(* Logix 5000 project; controller GEA_Test_Chamber vendor 1 type 14 code 196 rev 32.14; software revision 32.04; part 10 of 11 *)
(* tags used below, declared in another part *)
   bPulse1Hz : BOOL;
   Counter : COUNTER[20];
   LDO_LabView_Comm_OK : BOOL;
   LDO_Step : INT;
   LDO_Timer_Delay : TIMER[30];
   LDO_Water_Outlet_HighLimit : REAL;
   LDO_Water_Outlet_LowLimit : REAL;
   Oil_spray_11_ccmin : BOOL;
   ONS : BOOL[32];
   test : BOOL;
   Water_Outlet_Temp_OK : BOOL;
   Amount_Water_Flow : DINT;
   Client_01 : raC_Opr_NetModbusTCPClient;
   Client_01_Data : raC_UDT_ModbusClientData;
   Client_01_EN : BOOL;
   Client_01_MSG_Connect : MESSAGE;
   Client_01_MSG_Create : MESSAGE;
   Client_01_MSG_Delete : MESSAGE;
   Client_01_MSG_Read : MESSAGE;
   Client_01_MSG_SetSing : MESSAGE;
   Client_01_MSG_Write : MESSAGE;
   Client_01_Parameters : raC_UDT_ModbusClientConnection;
   Client_01_Transactions : raC_UDT_ModbusClientTransaction[5];
   Client_02 : raC_Opr_NetModbusTCPClient;
   Client_02_Data : raC_UDT_ModbusClientData;
   Client_02_EN : BOOL;
   Client_02_MSG_Connect : MESSAGE;
   Client_02_MSG_Create : MESSAGE;
   Client_02_MSG_Delete : MESSAGE;
   Client_02_MSG_Read : MESSAGE;
   Client_02_MSG_SetSing : MESSAGE;
   Client_02_MSG_Write : MESSAGE;
   Client_02_Parameters : raC_UDT_ModbusClientConnection;
   Client_02_Transactions : raC_UDT_ModbusClientTransaction[5];
   FVIR_Error_MSG : INT;
   FVIR_LabView_Control : INT;
   FVIR_LabView_Status : INT;
   FVIR_Mannequin_Direction_TimeDelay : INT;
   FVIR_Mannequin_Time_Pause : INT;
   FVIR_Number_Mannequin_Movement : INT;
   FVIR_Rate_REAL : REAL;
   FVIR_Reset_Cnt : BOOL;
   FVIR_Reset_Cnt_inprogress : BOOL;
   FVIR_Test_No : INT;
   FVIR_Totalizer_REAL : REAL;
   FVIR_Water_Flow_DRK375 : INT;
   FVIR_Water_Flow_DRK375_Float : REAL;
   FVIR_Water_Outlet_Valve : INT;
   FVIR_Water_Outlet_Valve_Flow_SP : REAL;
   FVIR_Water_Outlet_Valve_SP : REAL;
   FVIR_Water_Temp_DRK375 : INT;
   FVIR_Water_Temp_DRK375_Float : REAL;
   LDO_BurnerCycle_11_12_OFF : INT;
   LDO_BurnerCycle_11_12_ON : INT;
   LDO_BurnerCycle_13_OFF : INT;
   LDO_BurnerCycle_13_ON : INT;
   LDO_BurnerCycle_1_10_OFF : INT;
   LDO_BurnerCycle_1_10_ON : INT;
   LDO_Error_MSG : INT;
   LDO_LabView_Control : INT;
   LDO_LabView_Control2 : INT;
   LDO_LabView_Status : INT;
   LDO_Oil_1st_seq_OFF : INT;
   LDO_Oil_1st_seq_ON : INT;
   LDO_Oil_all_seq_OFF : INT;
   LDO_Oil_all_seq_ON : INT;
   LDO_Oil_pre_seq_OFF : INT;
   LDO_Oil_pre_seq_ON : INT;
   LDO_Reset_Cnt : BOOL;
   LDO_Reset_CNT_inprogress : BOOL;
   LDO_Water_Flow_DRK375_Float : REAL;
   LDO_Water_Outlet_Valve : REAL;
   LDO_Water_Outlet_Valve_Flow_SP : REAL;
   LDO_Water_Outlet_Valve_SP : REAL;
   LDO_Water_Temp_DRK375_Float : REAL;
   Modbus_LabView : raC_Opr_NetModbusTCPServer;
   Modbus_LabView_Data : raC_UDT_ModbusServerData;
   nLDO_Rate_REAL : REAL;
   nLDO_Totalizer_REAL : REAL;
   Output_LDO : Output_LDO;
   pulsReset : BOOL;
   SET_0 : BOOL;
   Timer_Delay_Start : TIMER;
(* LDO_Chamber, continued *)

ROUTINE LDO_Test   (* ladder *)
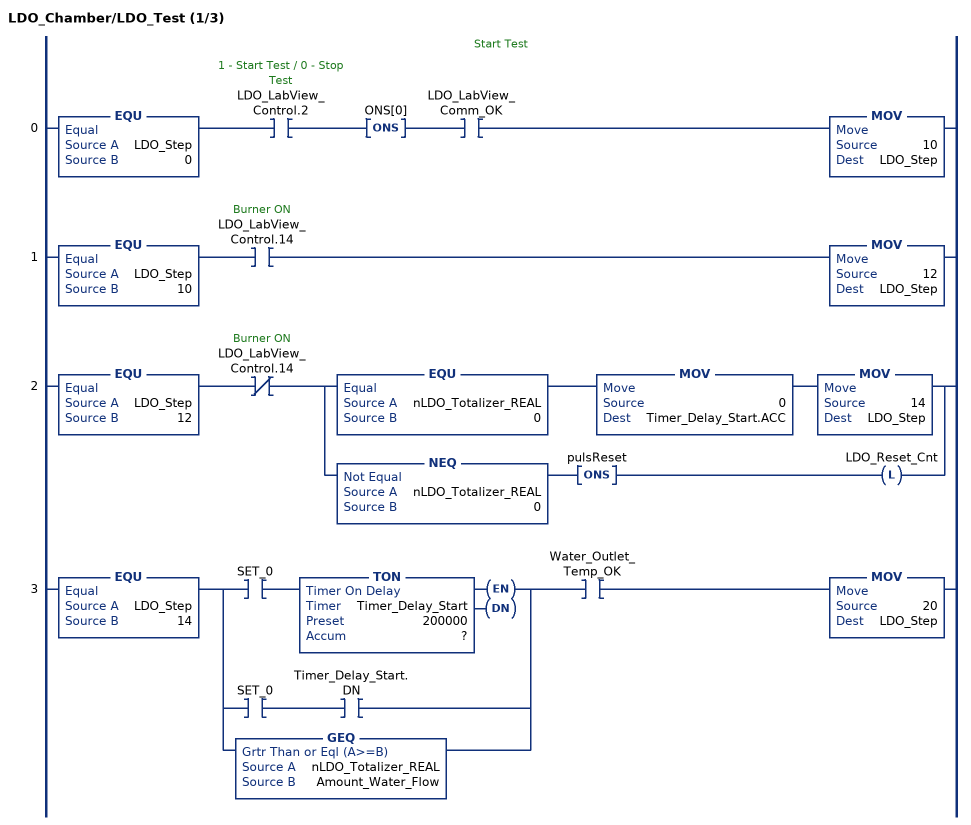
   // Start Test
   0: EQU(LDO_Step,0)XIC(LDO_LabView_Control.2)ONS(ONS[0])XIC(LDO_LabView_Comm_OK)MOV(10,LDO_Step);
   1: EQU(LDO_Step,10)XIC(LDO_LabView_Control.14)MOV(12,LDO_Step);
   2: EQU(LDO_Step,12)XIO(LDO_LabView_Control.14)[EQU(nLDO_Totalizer_REAL,0) MOV(0,Timer_Delay_Start.ACC) MOV(14,LDO_Step) ,NEQ(nLDO_Totalizer_REAL,0) ONS(pulsReset) OTL(LDO_Reset_Cnt) ];
   3: EQU(LDO_Step,14)[XIC(SET_0) TON(Timer_Delay_Start,?,?) ,XIC(SET_0) XIC(Timer_Delay_Start.DN) ,GEQ(nLDO_Totalizer_REAL,Amount_Water_Flow) ]XIC(Water_Outlet_Temp_OK)MOV(20,LDO_Step);
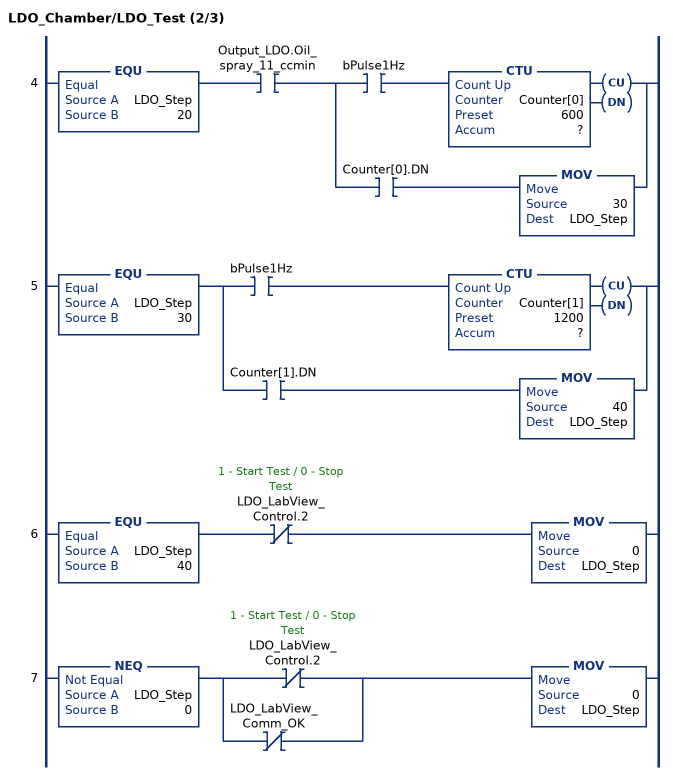
   4: EQU(LDO_Step,20)XIC(Output_LDO.Oil_spray_11_ccmin)[XIC(bPulse1Hz) CTU(Counter[0],?,?) ,XIC(Counter[0].DN) MOV(30,LDO_Step) ];
   5: EQU(LDO_Step,30)[XIC(bPulse1Hz) CTU(Counter[1],?,?) ,XIC(Counter[1].DN) MOV(40,LDO_Step) ];
   6: EQU(LDO_Step,40)XIO(LDO_LabView_Control.2)MOV(0,LDO_Step);
   7: NEQ(LDO_Step,0)[XIO(LDO_LabView_Control.2) ,XIO(LDO_LabView_Comm_OK) ]MOV(0,LDO_Step);
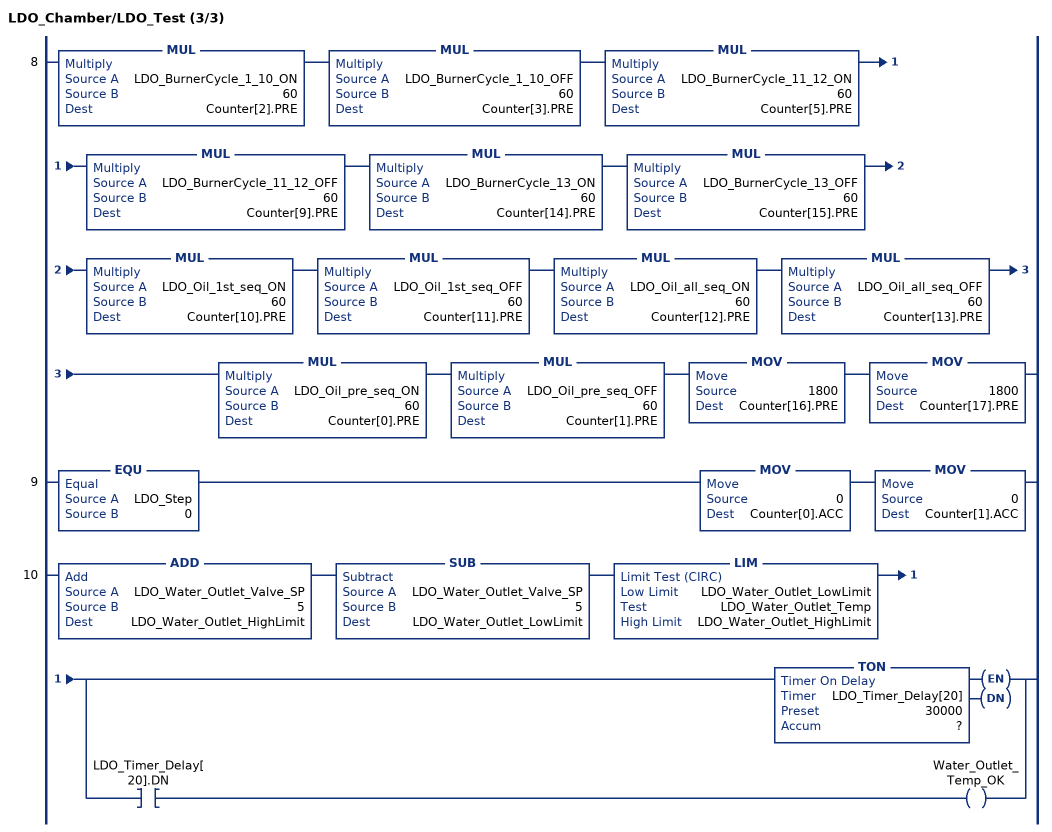
   8: MUL(LDO_BurnerCycle_1_10_ON,60,Counter[2].PRE)MUL(LDO_BurnerCycle_1_10_OFF,60,Counter[3].PRE)MUL(LDO_BurnerCycle_11_12_ON,60,Counter[5].PRE)MUL(LDO_BurnerCycle_11_12_OFF,60,Counter[9].PRE)MUL(LDO_BurnerCycle_13_ON,60,Counter[14].PRE)MUL(LDO_BurnerCycle_13_OFF,60,Counter[15].PRE)MUL(LDO_Oil_1st_seq_ON,60,Counter[10].PRE)MUL(LDO_Oil_1st_seq_OFF,60,Counter[11].PRE)MUL(LDO_Oil_all_seq_ON,60,Counter[12].PRE)MUL(LDO_Oil_all_seq_OFF,60,Counter[13].PRE)MUL(LDO_Oil_pre_seq_ON,60,Counter[0].PRE)MUL(LDO_Oil_pre_seq_OFF,60,Counter[1].PRE)MOV(1800,Counter[16].PRE)MOV(1800,Counter[17].PRE);
   9: EQU(LDO_Step,0)MOV(0,Counter[0].ACC)MOV(0,Counter[1].ACC);
   10: ADD(LDO_Water_Outlet_Valve_SP,5,LDO_Water_Outlet_HighLimit)SUB(LDO_Water_Outlet_Valve_SP,5,LDO_Water_Outlet_LowLimit)LIM(LDO_Water_Outlet_LowLimit,LDO_Water_Outlet_Temp,LDO_Water_Outlet_HighLimit)[TON(LDO_Timer_Delay[20],?,?) ,XIC(LDO_Timer_Delay[20].DN) OTE(Water_Outlet_Temp_OK) ];
END_ROUTINE
END_PROGRAM

PROGRAM Modbus_Client   (* main routine Main *)
VAR
   FVIR_Cnt_Reset : BOOL;
   FVIR_Rate_DINT : DINT;
   FVIR_Rate_value_temp : DINT;
   FVIR_Reset_Cnt_Timeout : TIMER := (PRE := 3000);
   FVIR_Reset_Cycle : DINT;
   FVIR_Timer_Delay_Reset : TIMER := (PRE := 500);
   FVIR_Timer_Reset : TIMER := (PRE := 500);
   FVIR_Total_DINT : DINT;
   FVIR_Total_value_temp : DINT;
   LDO_Cnt_Reset : BOOL;
   LDO_Rate_DINT : DINT;
   LDO_Rate_REAL : REAL;
   LDO_Rate_value_temp : DINT;
   LDO_Total_value_temp : DINT := 124780544;
   LDO_Totalizer_DINT : DINT := 1904;
   LDO_Totalizer_REAL : REAL := 4.91;
   LDO_Valley_value : DINT := 2034;
   LDO_Valley_value_temp : DINT := 133300224;
   Modbus_FVIR_Off : BOOL := 1;
   nLDO_Total_Mem : REAL := 565.7;
   off : BOOL := 1;
   ONS_1 : BOOL := 1;
   ONS_2 : BOOL;
   Reset_Cnt_Timeout : TIMER := (PRE := 3000);
   Reset_Cycle : DINT;
   Timer_Delay_Reset : TIMER := (PRE := 500);
   Timer_Reset : TIMER := (PRE := 500);
END_VAR

ROUTINE FVIR_Flow_Outlet_Meter   (* ladder *)
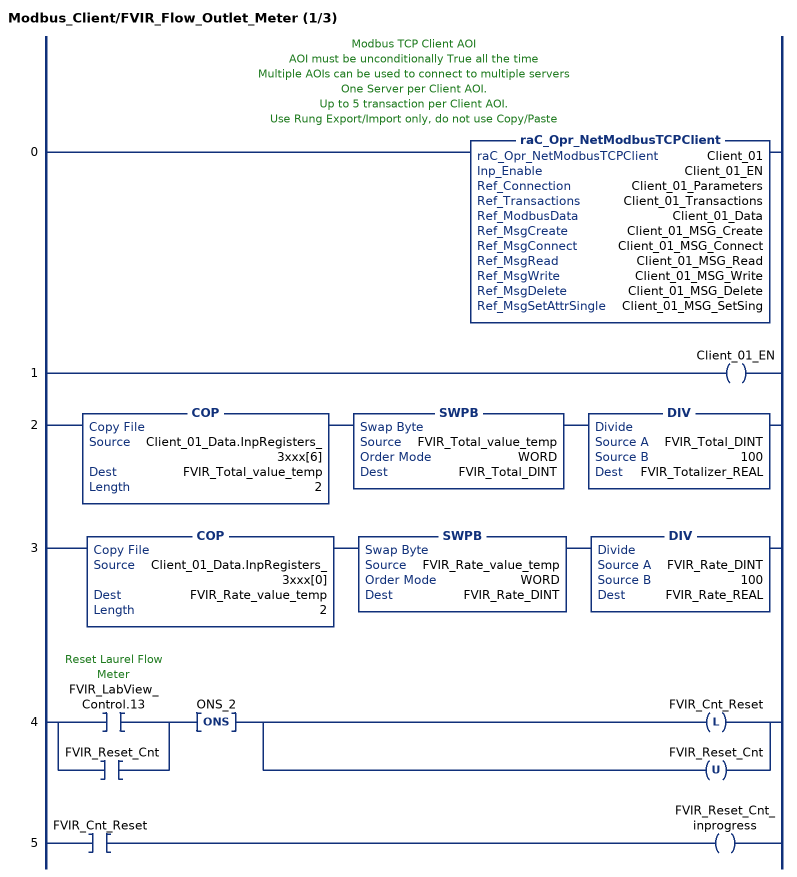
   // Modbus TCP Client AOI
   // AOI must be unconditionally True all the time
   // Multiple AOIs can be used to connect to multiple servers
   // One Server per Client AOI.
   //  Up to 5 transaction per Client AOI.
   // Use Rung Export/Import only, do not use Copy/Paste
   0: raC_Opr_NetModbusTCPClient(Client_01,Client_01_EN,Client_01_Parameters,Client_01_Transactions,Client_01_Data,Client_01_MSG_Create,Client_01_MSG_Connect,Client_01_MSG_Read,Client_01_MSG_Write,Client_01_MSG_Delete,Client_01_MSG_SetSing);
   1: OTE(Client_01_EN);
   2: COP(Client_01_Data.InpRegisters_3xxx[6],FVIR_Total_value_temp,2)SWPB(FVIR_Total_value_temp,WORD,FVIR_Total_DINT)DIV(FVIR_Total_DINT,100,FVIR_Totalizer_REAL);
   3: COP(Client_01_Data.InpRegisters_3xxx[0],FVIR_Rate_value_temp,2)SWPB(FVIR_Rate_value_temp,WORD,FVIR_Rate_DINT)DIV(FVIR_Rate_DINT,100,FVIR_Rate_REAL);
   4: [XIC(FVIR_LabView_Control.13) ,XIC(FVIR_Reset_Cnt) ]ONS(ONS_2)[OTL(FVIR_Cnt_Reset) ,OTU(FVIR_Reset_Cnt) ];
   5: XIC(FVIR_Cnt_Reset)OTE(FVIR_Reset_Cnt_inprogress);
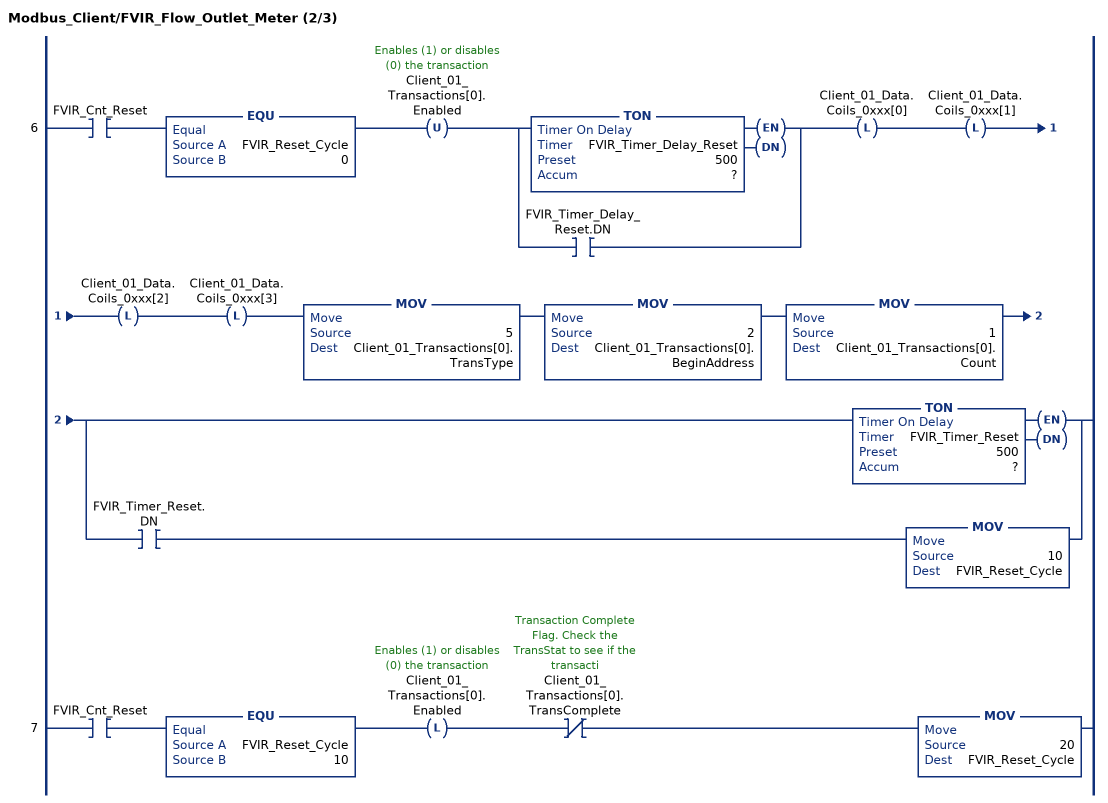
   6: XIC(FVIR_Cnt_Reset)EQU(FVIR_Reset_Cycle,0)OTU(Client_01_Transactions[0].Enabled)[TON(FVIR_Timer_Delay_Reset,?,?) ,XIC(FVIR_Timer_Delay_Reset.DN) ]OTL(Client_01_Data.Coils_0xxx[0])OTL(Client_01_Data.Coils_0xxx[1])OTL(Client_01_Data.Coils_0xxx[2])OTL(Client_01_Data.Coils_0xxx[3])MOV(5,Client_01_Transactions[0].TransType)MOV(2,Client_01_Transactions[0].BeginAddress)MOV(1,Client_01_Transactions[0].Count)[TON(FVIR_Timer_Reset,?,?) ,XIC(FVIR_Timer_Reset.DN) MOV(10,FVIR_Reset_Cycle) ];
   7: XIC(FVIR_Cnt_Reset)EQU(FVIR_Reset_Cycle,10)OTL(Client_01_Transactions[0].Enabled)XIO(Client_01_Transactions[0].TransComplete)MOV(20,FVIR_Reset_Cycle);
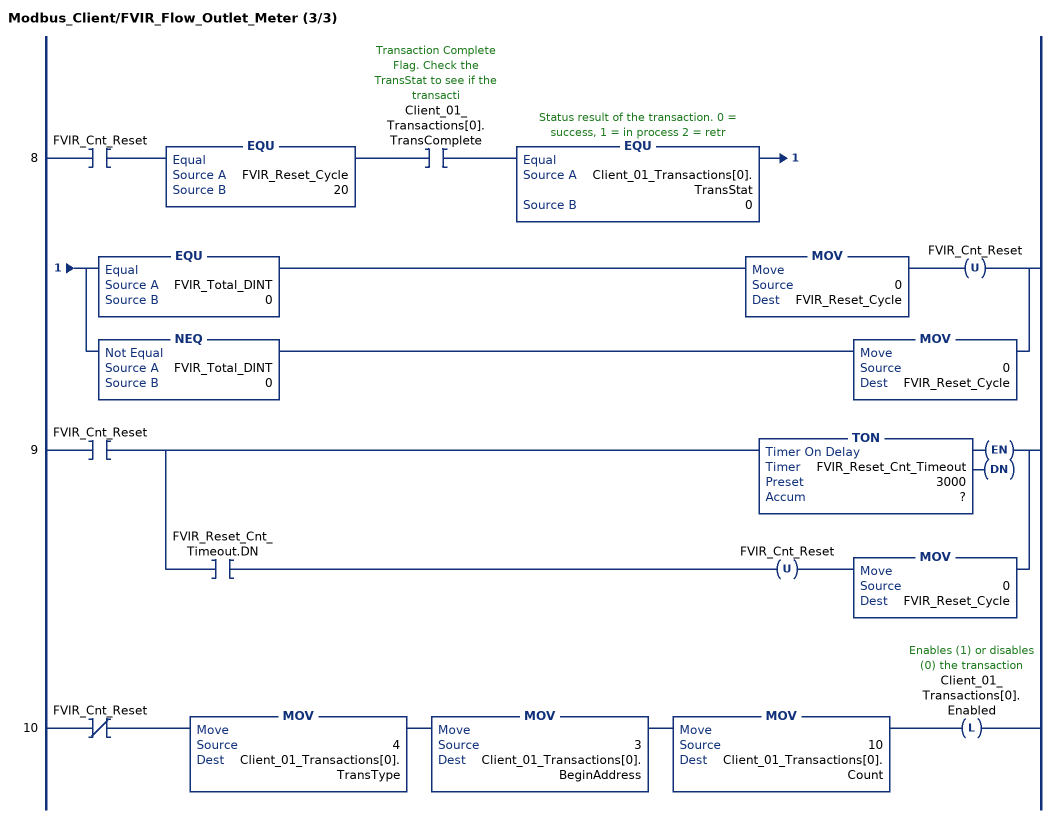
   8: XIC(FVIR_Cnt_Reset)EQU(FVIR_Reset_Cycle,20)XIC(Client_01_Transactions[0].TransComplete)EQU(Client_01_Transactions[0].TransStat,0)[EQU(FVIR_Total_DINT,0) MOV(0,FVIR_Reset_Cycle) OTU(FVIR_Cnt_Reset) ,NEQ(FVIR_Total_DINT,0) MOV(0,FVIR_Reset_Cycle) ];
   9: XIC(FVIR_Cnt_Reset)[TON(FVIR_Reset_Cnt_Timeout,?,?) ,XIC(FVIR_Reset_Cnt_Timeout.DN) OTU(FVIR_Cnt_Reset) MOV(0,FVIR_Reset_Cycle) ];
   10: XIO(FVIR_Cnt_Reset)MOV(4,Client_01_Transactions[0].TransType)MOV(3,Client_01_Transactions[0].BeginAddress)MOV(10,Client_01_Transactions[0].Count)OTL(Client_01_Transactions[0].Enabled);
END_ROUTINE

ROUTINE LDO_Flow_Outlet_Meter   (* ladder *)
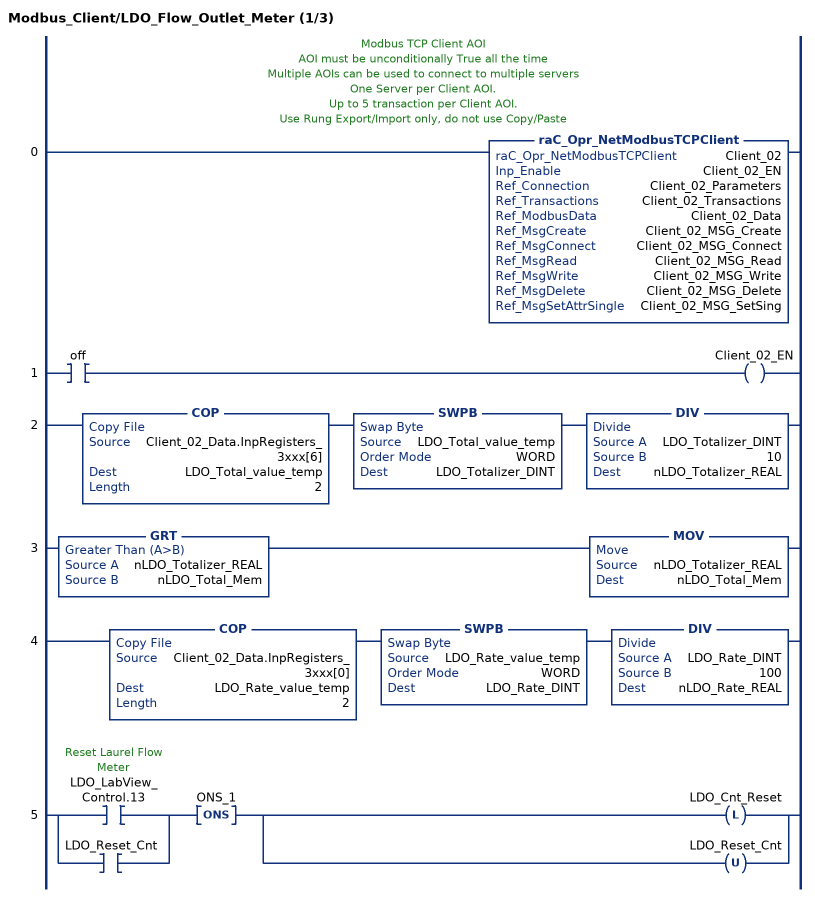
   // Modbus TCP Client AOI
   // AOI must be unconditionally True all the time
   // Multiple AOIs can be used to connect to multiple servers
   // One Server per Client AOI.
   //  Up to 5 transaction per Client AOI.
   // Use Rung Export/Import only, do not use Copy/Paste
   0: raC_Opr_NetModbusTCPClient(Client_02,Client_02_EN,Client_02_Parameters,Client_02_Transactions,Client_02_Data,Client_02_MSG_Create,Client_02_MSG_Connect,Client_02_MSG_Read,Client_02_MSG_Write,Client_02_MSG_Delete,Client_02_MSG_SetSing);
   1: XIC(off)OTE(Client_02_EN);
   2: COP(Client_02_Data.InpRegisters_3xxx[6],LDO_Total_value_temp,2)SWPB(LDO_Total_value_temp,WORD,LDO_Totalizer_DINT)DIV(LDO_Totalizer_DINT,10,nLDO_Totalizer_REAL);
   3: GRT(nLDO_Totalizer_REAL,nLDO_Total_Mem)MOV(nLDO_Totalizer_REAL,nLDO_Total_Mem);
   4: COP(Client_02_Data.InpRegisters_3xxx[0],LDO_Rate_value_temp,2)SWPB(LDO_Rate_value_temp,WORD,LDO_Rate_DINT)DIV(LDO_Rate_DINT,100,nLDO_Rate_REAL);
   5: [XIC(LDO_LabView_Control.13) ,XIC(LDO_Reset_Cnt) ]ONS(ONS_1)[OTL(LDO_Cnt_Reset) ,OTU(LDO_Reset_Cnt) ];
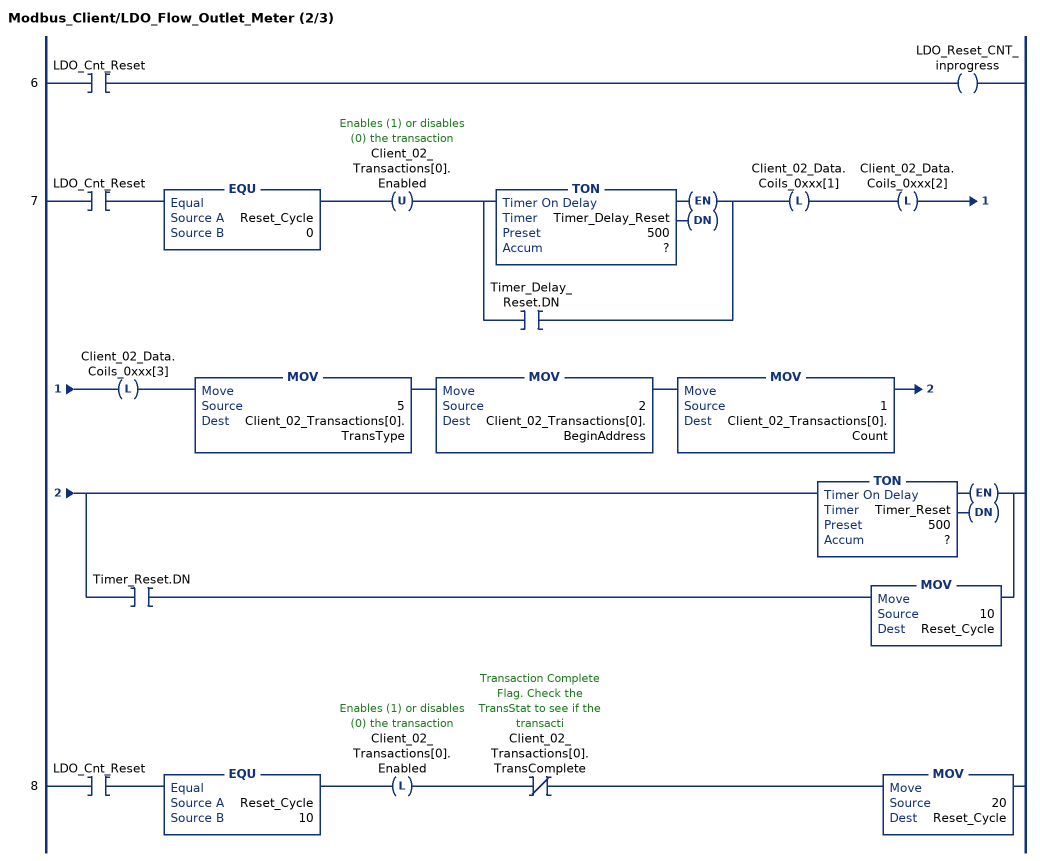
   6: XIC(LDO_Cnt_Reset)OTE(LDO_Reset_CNT_inprogress);
   7: XIC(LDO_Cnt_Reset)EQU(Reset_Cycle,0)OTU(Client_02_Transactions[0].Enabled)[TON(Timer_Delay_Reset,?,?) ,XIC(Timer_Delay_Reset.DN) ]OTL(Client_02_Data.Coils_0xxx[1])OTL(Client_02_Data.Coils_0xxx[2])OTL(Client_02_Data.Coils_0xxx[3])MOV(5,Client_02_Transactions[0].TransType)MOV(2,Client_02_Transactions[0].BeginAddress)MOV(1,Client_02_Transactions[0].Count)[TON(Timer_Reset,?,?) ,XIC(Timer_Reset.DN) MOV(10,Reset_Cycle) ];
   8: XIC(LDO_Cnt_Reset)EQU(Reset_Cycle,10)OTL(Client_02_Transactions[0].Enabled)XIO(Client_02_Transactions[0].TransComplete)MOV(20,Reset_Cycle);
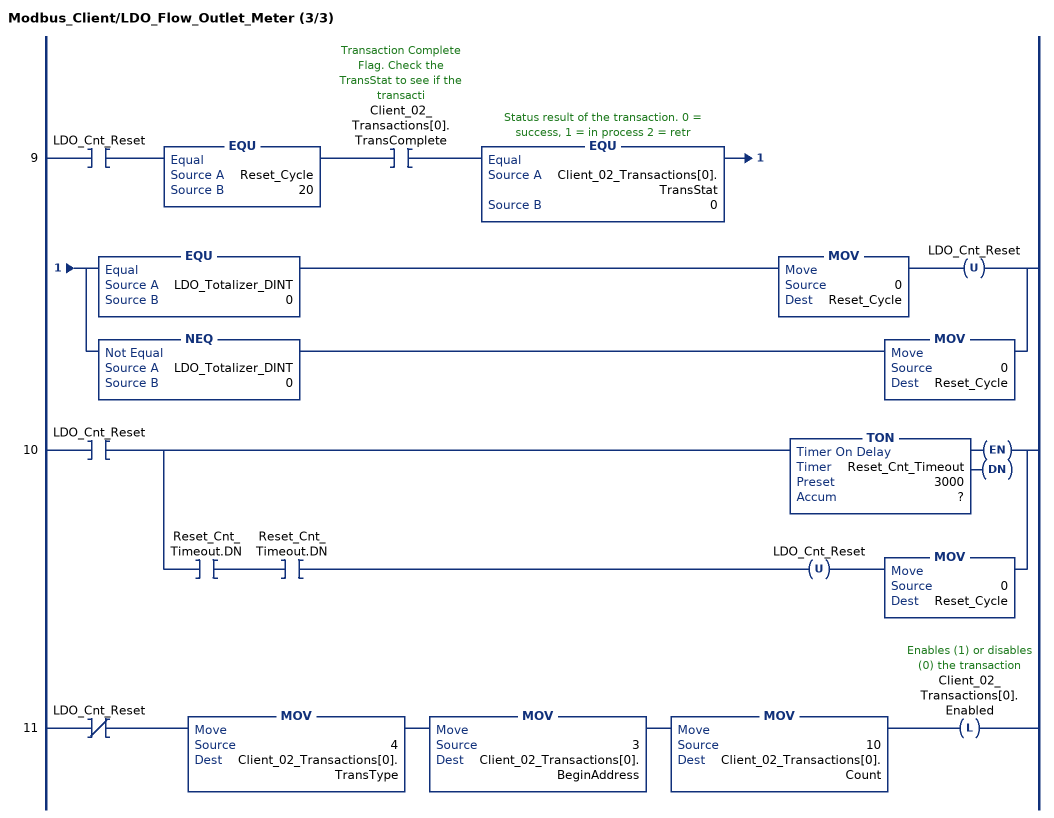
   9: XIC(LDO_Cnt_Reset)EQU(Reset_Cycle,20)XIC(Client_02_Transactions[0].TransComplete)EQU(Client_02_Transactions[0].TransStat,0)[EQU(LDO_Totalizer_DINT,0) MOV(0,Reset_Cycle) OTU(LDO_Cnt_Reset) ,NEQ(LDO_Totalizer_DINT,0) MOV(0,Reset_Cycle) ];
   10: XIC(LDO_Cnt_Reset)[TON(Reset_Cnt_Timeout,?,?) ,XIC(Reset_Cnt_Timeout.DN) XIC(Reset_Cnt_Timeout.DN) OTU(LDO_Cnt_Reset) MOV(0,Reset_Cycle) ];
   11: XIO(LDO_Cnt_Reset)MOV(4,Client_02_Transactions[0].TransType)MOV(3,Client_02_Transactions[0].BeginAddress)MOV(10,Client_02_Transactions[0].Count)OTL(Client_02_Transactions[0].Enabled);
END_ROUTINE

ROUTINE Main   (* ladder *)
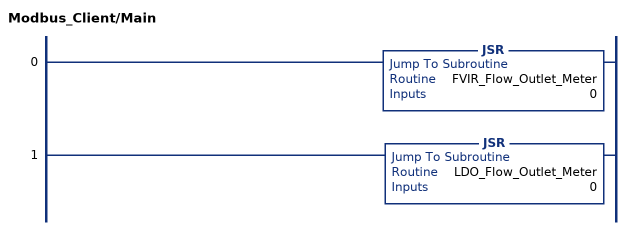
   0: JSR(FVIR_Flow_Outlet_Meter,0);
   1: JSR(LDO_Flow_Outlet_Meter,0);
END_ROUTINE
END_PROGRAM

PROGRAM Modbus_LabView   (* main routine Main *)
VAR
   DateTime : DINT[6];
   Empty : DINT;
   FVIR_SWPB_Data_Input : INT[10];
   FVIR_SWPB_Data_Output : INT[30] := ([0] := 8449, [1] := -32000, [2] := 2563);
   FVIR_SWPB_Data_Output_DINT : DINT[30];
   FVIR_TC : INT[30] := ([0] := 695, [1] := 689, [2] := 688, [3] := 698, [4] := 898, [5] := 859, [6] := 678, [7] := -1495, [8] := 671, [9] := 1181, [10] := -3497, [11] := -3470, [12] := -3508, [13] := -3483, [14] := -3499, [15] := -3480, [16] := -3290, [17] := -3270, [18] := -3280, [19] := -3275, [20] := 684, [21] := 684, [22] := 691, [23] := 681, [24] := 1000, [25] := 288, [26] := -50, [27] := -50);
   LDO_SWPB_Data_Input : INT[30];
   LDO_SWPB_Data_Output : INT[30] := ([0] := 256, [1] := -32000, [2] := 8456, [3] := 32256);
   LDO_SWPB_Data_Output_DINT : DINT[30];
   LDO_Water_Outlet_Temp : INT;
   Mod_Serv_On : BOOL;
   ModbusTCPIP_Data_SWPB : INT[100] := ([0] := 10038, [1] := 9949, [2] := 10074, [3] := 9937, [4] := 10433, [5] := 10296, [6] := 10421, [7] := 10237, [8] := 30936, [9] := 30936, [10] := 30936, [11] := 30936, [12] := 30936, [13] := 30936, [14] := 30936, [15] := 30936, [16] := 32736, [17] := 32736, [18] := 32736, [19] := 32736, [20] := 5450, [21] := 5700, [22] := 5490, [23] := 5750, [24] := 10500, [25] := 10500, [30] := 9664, [31] := 9664, [32] := 9664, [33] := 9664, [34] := 9664, [35] := 9664, [36] := 10500, [37] := 10500, [38] := 9664, [39] := 9664, [40] := 22592, [41] := 22592, [42] := 22592, [43] := 22592, [44] := -11984, [45] := -11984, [46] := 9664, [47] := 9664, [48] := 10500, [49] := 10500, [50] := 10500, [51] := 10500, [53] := 3916);
   New_MBTCP : BOOL := 1;
   Reserve : INT;
   TC : INT[30] := ([0] := 1007, [1] := 956, [2] := 730, [3] := 776, [4] := 729, [5] := 728, [6] := 724, [7] := 720, [8] := 741, [9] := 744, [10] := 1356, [11] := 21870, [12] := 21870, [13] := 21870, [14] := 24966, [15] := 24966, [16] := 24966, [17] := 24966);
        [25]   // Local Tag for Water Pressure Sensor FVIR (Not used currently)
END_VAR

ROUTINE Main   (* ladder *)
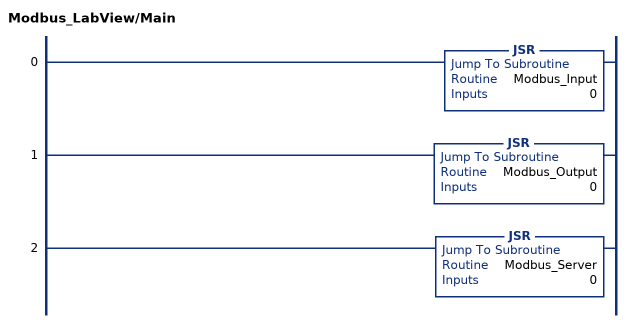
   0: JSR(Modbus_Input,0);
   1: JSR(Modbus_Output,0);
   2: JSR(Modbus_Server,0);
END_ROUTINE

ROUTINE Modbus_Input   (* ladder *)
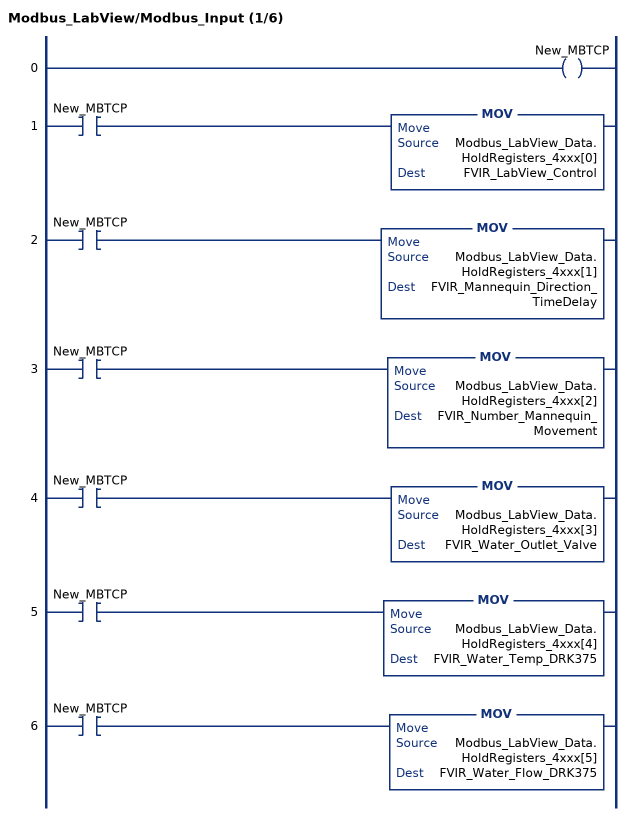
   0: OTE(New_MBTCP);
   1: XIC(New_MBTCP)MOV(Modbus_LabView_Data.HoldRegisters_4xxx[0],FVIR_LabView_Control);
   2: XIC(New_MBTCP)MOV(Modbus_LabView_Data.HoldRegisters_4xxx[1],FVIR_Mannequin_Direction_TimeDelay);
   3: XIC(New_MBTCP)MOV(Modbus_LabView_Data.HoldRegisters_4xxx[2],FVIR_Number_Mannequin_Movement);
   4: XIC(New_MBTCP)MOV(Modbus_LabView_Data.HoldRegisters_4xxx[3],FVIR_Water_Outlet_Valve);
   5: XIC(New_MBTCP)MOV(Modbus_LabView_Data.HoldRegisters_4xxx[4],FVIR_Water_Temp_DRK375);
   6: XIC(New_MBTCP)MOV(Modbus_LabView_Data.HoldRegisters_4xxx[5],FVIR_Water_Flow_DRK375);
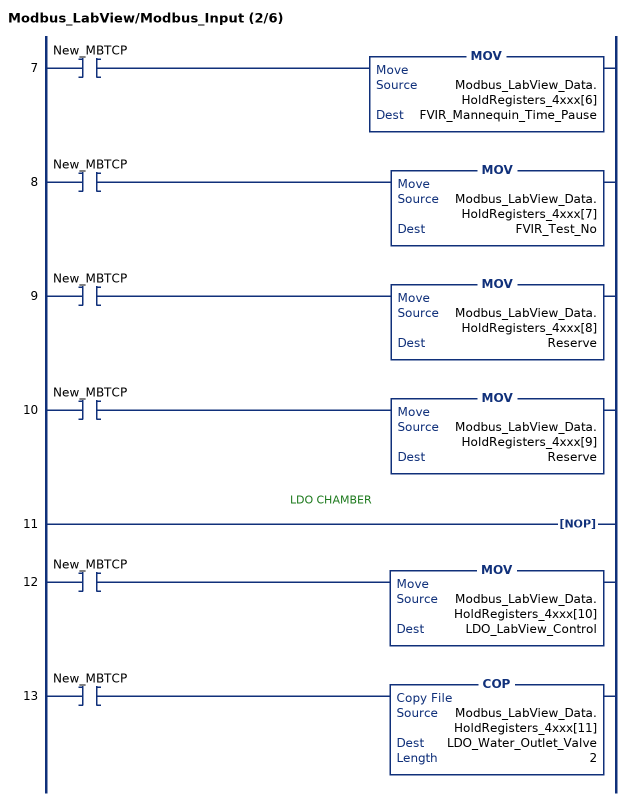
   7: XIC(New_MBTCP)MOV(Modbus_LabView_Data.HoldRegisters_4xxx[6],FVIR_Mannequin_Time_Pause);
   8: XIC(New_MBTCP)MOV(Modbus_LabView_Data.HoldRegisters_4xxx[7],FVIR_Test_No);
   9: XIC(New_MBTCP)MOV(Modbus_LabView_Data.HoldRegisters_4xxx[8],Reserve);
   10: XIC(New_MBTCP)MOV(Modbus_LabView_Data.HoldRegisters_4xxx[9],Reserve);
   // LDO CHAMBER
   11: NOP();
   12: XIC(New_MBTCP)MOV(Modbus_LabView_Data.HoldRegisters_4xxx[10],LDO_LabView_Control);
   13: XIC(New_MBTCP)COP(Modbus_LabView_Data.HoldRegisters_4xxx[11],LDO_Water_Outlet_Valve,2);
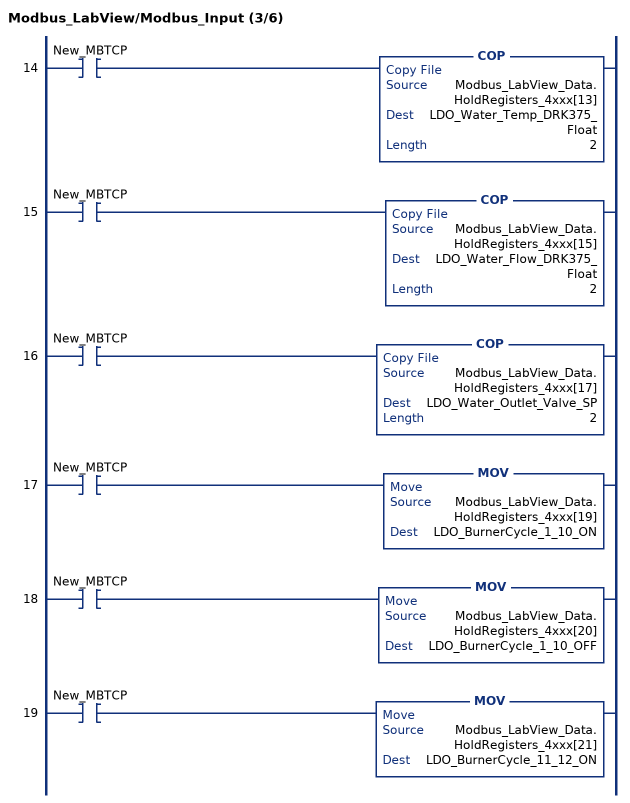
   14: XIC(New_MBTCP)COP(Modbus_LabView_Data.HoldRegisters_4xxx[13],LDO_Water_Temp_DRK375_Float,2);
   15: XIC(New_MBTCP)COP(Modbus_LabView_Data.HoldRegisters_4xxx[15],LDO_Water_Flow_DRK375_Float,2);
   16: XIC(New_MBTCP)COP(Modbus_LabView_Data.HoldRegisters_4xxx[17],LDO_Water_Outlet_Valve_SP,2);
   17: XIC(New_MBTCP)MOV(Modbus_LabView_Data.HoldRegisters_4xxx[19],LDO_BurnerCycle_1_10_ON);
   18: XIC(New_MBTCP)MOV(Modbus_LabView_Data.HoldRegisters_4xxx[20],LDO_BurnerCycle_1_10_OFF);
   19: XIC(New_MBTCP)MOV(Modbus_LabView_Data.HoldRegisters_4xxx[21],LDO_BurnerCycle_11_12_ON);
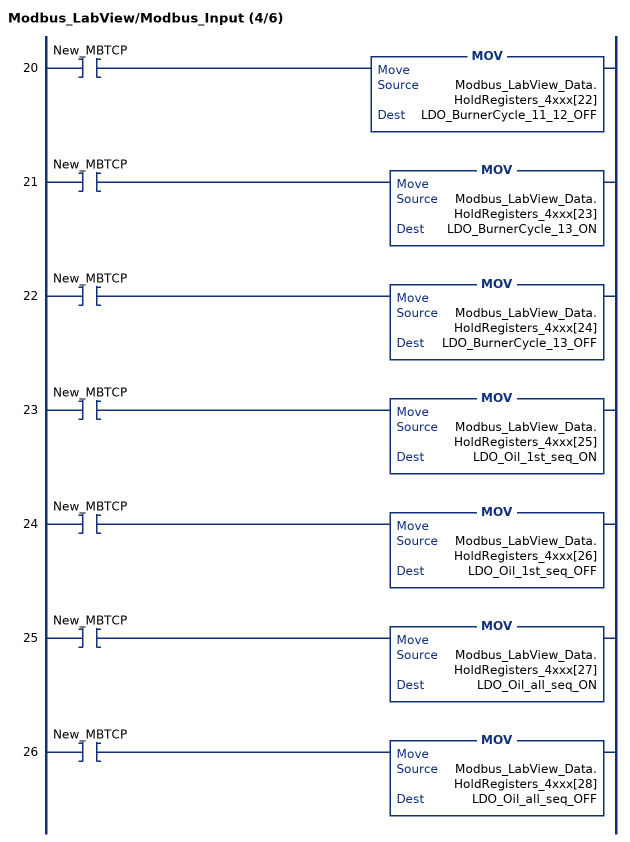
   20: XIC(New_MBTCP)MOV(Modbus_LabView_Data.HoldRegisters_4xxx[22],LDO_BurnerCycle_11_12_OFF);
   21: XIC(New_MBTCP)MOV(Modbus_LabView_Data.HoldRegisters_4xxx[23],LDO_BurnerCycle_13_ON);
   22: XIC(New_MBTCP)MOV(Modbus_LabView_Data.HoldRegisters_4xxx[24],LDO_BurnerCycle_13_OFF);
   23: XIC(New_MBTCP)MOV(Modbus_LabView_Data.HoldRegisters_4xxx[25],LDO_Oil_1st_seq_ON);
   24: XIC(New_MBTCP)MOV(Modbus_LabView_Data.HoldRegisters_4xxx[26],LDO_Oil_1st_seq_OFF);
   25: XIC(New_MBTCP)MOV(Modbus_LabView_Data.HoldRegisters_4xxx[27],LDO_Oil_all_seq_ON);
   26: XIC(New_MBTCP)MOV(Modbus_LabView_Data.HoldRegisters_4xxx[28],LDO_Oil_all_seq_OFF);
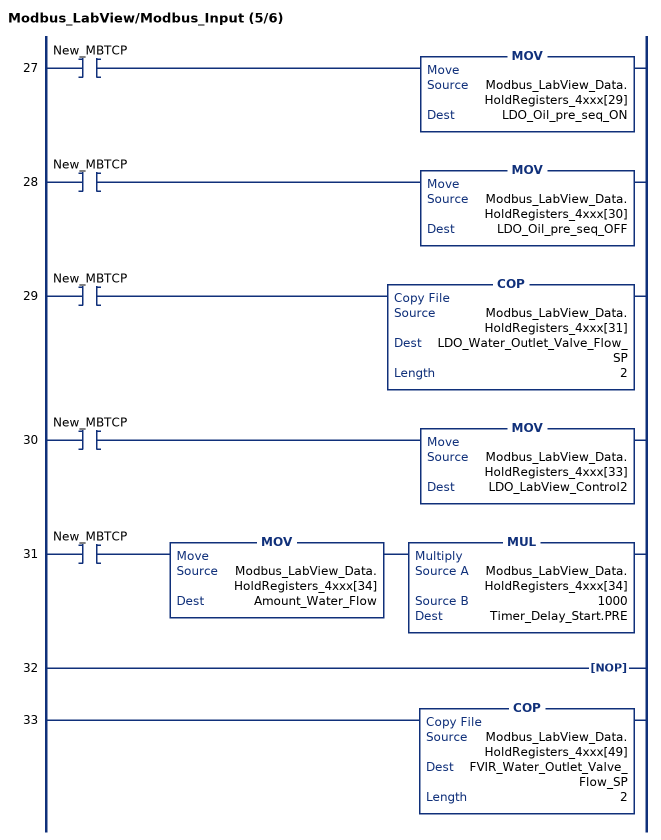
   27: XIC(New_MBTCP)MOV(Modbus_LabView_Data.HoldRegisters_4xxx[29],LDO_Oil_pre_seq_ON);
   28: XIC(New_MBTCP)MOV(Modbus_LabView_Data.HoldRegisters_4xxx[30],LDO_Oil_pre_seq_OFF);
   29: XIC(New_MBTCP)COP(Modbus_LabView_Data.HoldRegisters_4xxx[31],LDO_Water_Outlet_Valve_Flow_SP,2);
   30: XIC(New_MBTCP)MOV(Modbus_LabView_Data.HoldRegisters_4xxx[33],LDO_LabView_Control2);
   31: XIC(New_MBTCP)MOV(Modbus_LabView_Data.HoldRegisters_4xxx[34],Amount_Water_Flow)MUL(Modbus_LabView_Data.HoldRegisters_4xxx[34],1000,Timer_Delay_Start.PRE);
   32: NOP();
   33: COP(Modbus_LabView_Data.HoldRegisters_4xxx[49],FVIR_Water_Outlet_Valve_Flow_SP,2);
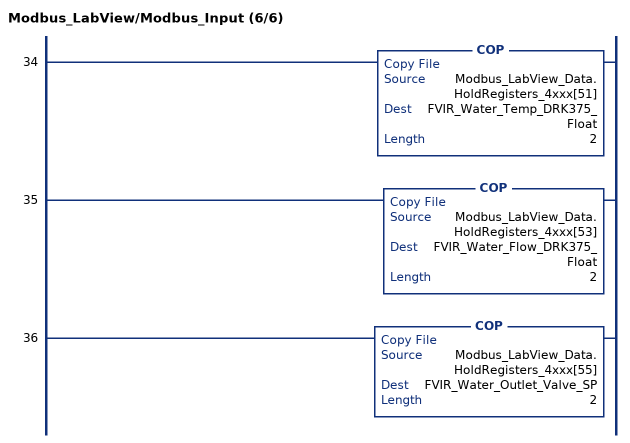
   34: COP(Modbus_LabView_Data.HoldRegisters_4xxx[51],FVIR_Water_Temp_DRK375_Float,2);
   35: COP(Modbus_LabView_Data.HoldRegisters_4xxx[53],FVIR_Water_Flow_DRK375_Float,2);
   36: COP(Modbus_LabView_Data.HoldRegisters_4xxx[55],FVIR_Water_Outlet_Valve_SP,2);
END_ROUTINE

ROUTINE Modbus_Output   (* ladder *)
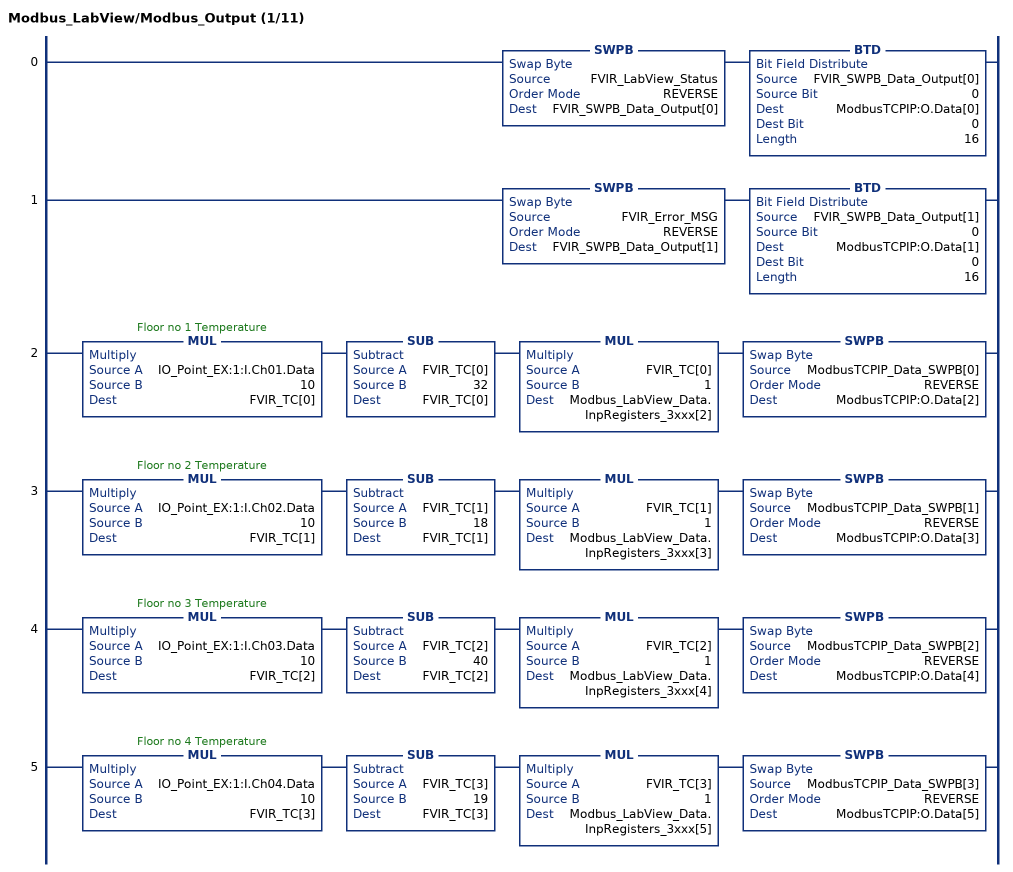
   0: SWPB(FVIR_LabView_Status,REVERSE,FVIR_SWPB_Data_Output[0])BTD(FVIR_SWPB_Data_Output[0],0,ModbusTCPIP:O.Data[0],0,16);
   1: SWPB(FVIR_Error_MSG,REVERSE,FVIR_SWPB_Data_Output[1])BTD(FVIR_SWPB_Data_Output[1],0,ModbusTCPIP:O.Data[1],0,16);
   2: MUL(IO_Point_EX:1:I.Ch01.Data,10,FVIR_TC[0])SUB(FVIR_TC[0],32,FVIR_TC[0])MUL(FVIR_TC[0],1,Modbus_LabView_Data.InpRegisters_3xxx[2])SWPB(ModbusTCPIP_Data_SWPB[0],REVERSE,ModbusTCPIP:O.Data[2]);
   3: MUL(IO_Point_EX:1:I.Ch02.Data,10,FVIR_TC[1])SUB(FVIR_TC[1],18,FVIR_TC[1])MUL(FVIR_TC[1],1,Modbus_LabView_Data.InpRegisters_3xxx[3])SWPB(ModbusTCPIP_Data_SWPB[1],REVERSE,ModbusTCPIP:O.Data[3]);
   4: MUL(IO_Point_EX:1:I.Ch03.Data,10,FVIR_TC[2])SUB(FVIR_TC[2],40,FVIR_TC[2])MUL(FVIR_TC[2],1,Modbus_LabView_Data.InpRegisters_3xxx[4])SWPB(ModbusTCPIP_Data_SWPB[2],REVERSE,ModbusTCPIP:O.Data[4]);
   5: MUL(IO_Point_EX:1:I.Ch04.Data,10,FVIR_TC[3])SUB(FVIR_TC[3],19,FVIR_TC[3])MUL(FVIR_TC[3],1,Modbus_LabView_Data.InpRegisters_3xxx[5])SWPB(ModbusTCPIP_Data_SWPB[3],REVERSE,ModbusTCPIP:O.Data[5]);
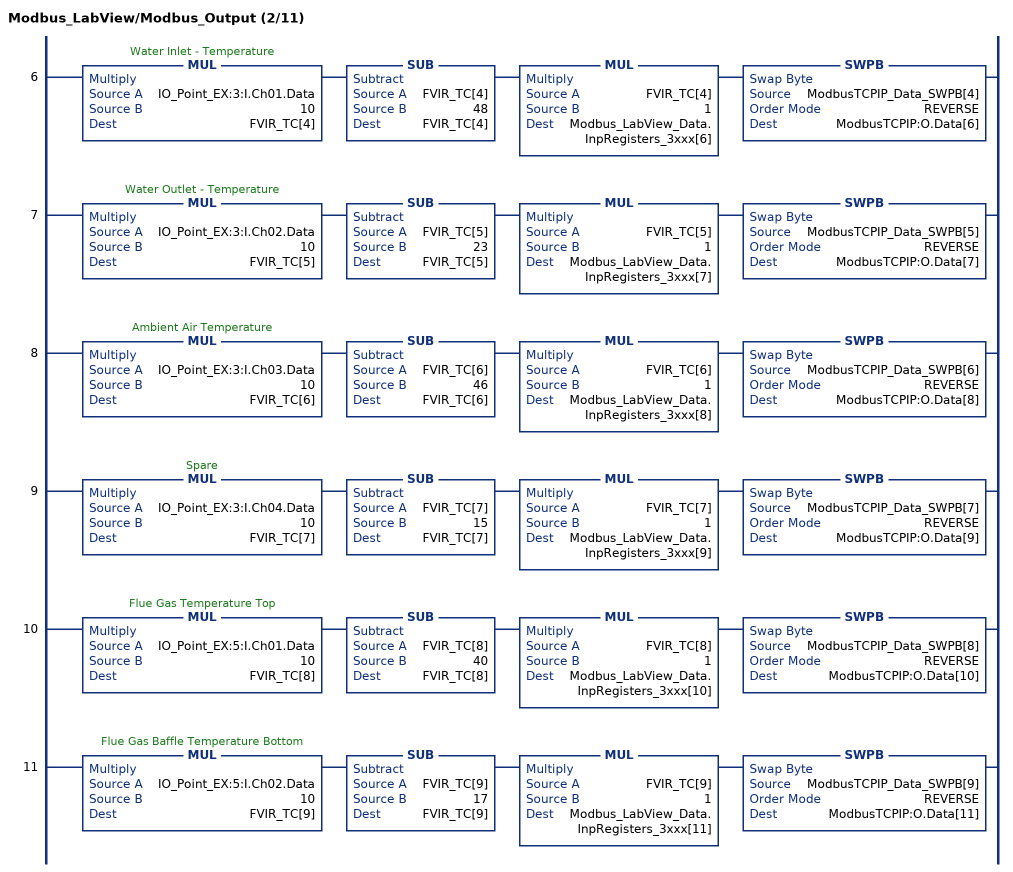
   6: MUL(IO_Point_EX:3:I.Ch01.Data,10,FVIR_TC[4])SUB(FVIR_TC[4],48,FVIR_TC[4])MUL(FVIR_TC[4],1,Modbus_LabView_Data.InpRegisters_3xxx[6])SWPB(ModbusTCPIP_Data_SWPB[4],REVERSE,ModbusTCPIP:O.Data[6]);
   7: MUL(IO_Point_EX:3:I.Ch02.Data,10,FVIR_TC[5])SUB(FVIR_TC[5],23,FVIR_TC[5])MUL(FVIR_TC[5],1,Modbus_LabView_Data.InpRegisters_3xxx[7])SWPB(ModbusTCPIP_Data_SWPB[5],REVERSE,ModbusTCPIP:O.Data[7]);
   8: MUL(IO_Point_EX:3:I.Ch03.Data,10,FVIR_TC[6])SUB(FVIR_TC[6],46,FVIR_TC[6])MUL(FVIR_TC[6],1,Modbus_LabView_Data.InpRegisters_3xxx[8])SWPB(ModbusTCPIP_Data_SWPB[6],REVERSE,ModbusTCPIP:O.Data[8]);
   9: MUL(IO_Point_EX:3:I.Ch04.Data,10,FVIR_TC[7])SUB(FVIR_TC[7],15,FVIR_TC[7])MUL(FVIR_TC[7],1,Modbus_LabView_Data.InpRegisters_3xxx[9])SWPB(ModbusTCPIP_Data_SWPB[7],REVERSE,ModbusTCPIP:O.Data[9]);
   10: MUL(IO_Point_EX:5:I.Ch01.Data,10,FVIR_TC[8])SUB(FVIR_TC[8],40,FVIR_TC[8])MUL(FVIR_TC[8],1,Modbus_LabView_Data.InpRegisters_3xxx[10])SWPB(ModbusTCPIP_Data_SWPB[8],REVERSE,ModbusTCPIP:O.Data[10]);
   11: MUL(IO_Point_EX:5:I.Ch02.Data,10,FVIR_TC[9])SUB(FVIR_TC[9],17,FVIR_TC[9])MUL(FVIR_TC[9],1,Modbus_LabView_Data.InpRegisters_3xxx[11])SWPB(ModbusTCPIP_Data_SWPB[9],REVERSE,ModbusTCPIP:O.Data[11]);
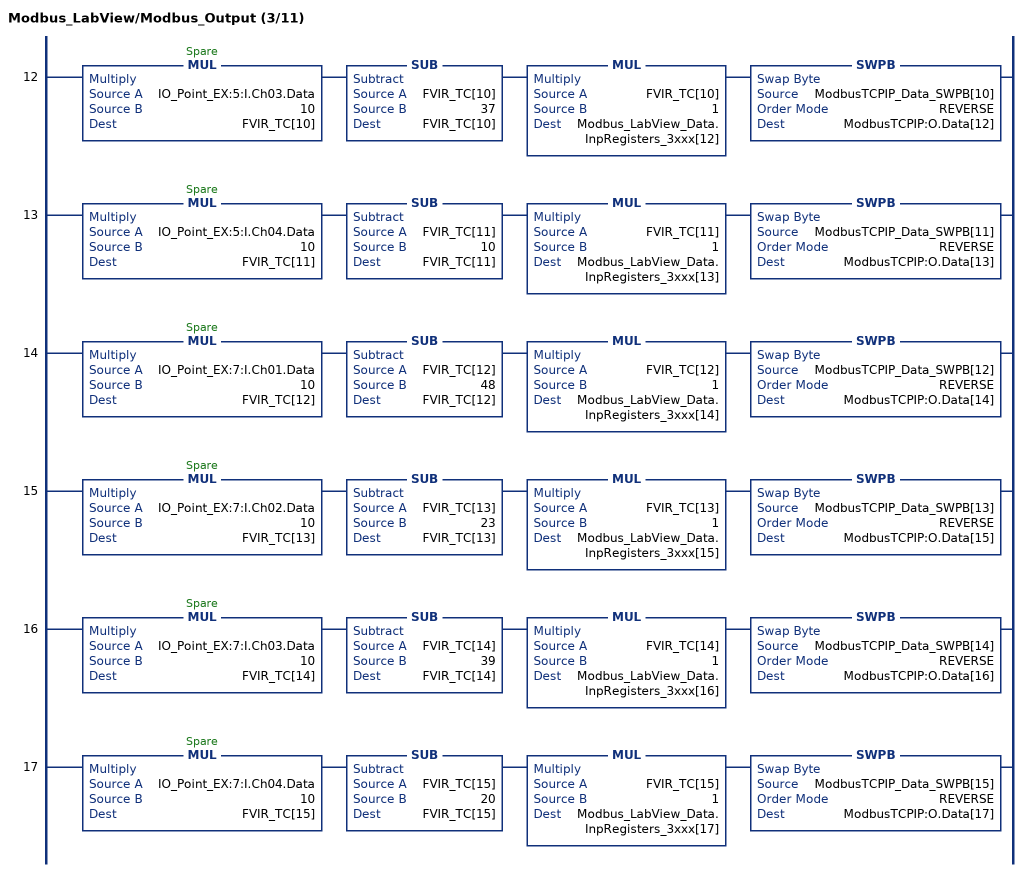
   12: MUL(IO_Point_EX:5:I.Ch03.Data,10,FVIR_TC[10])SUB(FVIR_TC[10],37,FVIR_TC[10])MUL(FVIR_TC[10],1,Modbus_LabView_Data.InpRegisters_3xxx[12])SWPB(ModbusTCPIP_Data_SWPB[10],REVERSE,ModbusTCPIP:O.Data[12]);
   13: MUL(IO_Point_EX:5:I.Ch04.Data,10,FVIR_TC[11])SUB(FVIR_TC[11],10,FVIR_TC[11])MUL(FVIR_TC[11],1,Modbus_LabView_Data.InpRegisters_3xxx[13])SWPB(ModbusTCPIP_Data_SWPB[11],REVERSE,ModbusTCPIP:O.Data[13]);
   14: MUL(IO_Point_EX:7:I.Ch01.Data,10,FVIR_TC[12])SUB(FVIR_TC[12],48,FVIR_TC[12])MUL(FVIR_TC[12],1,Modbus_LabView_Data.InpRegisters_3xxx[14])SWPB(ModbusTCPIP_Data_SWPB[12],REVERSE,ModbusTCPIP:O.Data[14]);
   15: MUL(IO_Point_EX:7:I.Ch02.Data,10,FVIR_TC[13])SUB(FVIR_TC[13],23,FVIR_TC[13])MUL(FVIR_TC[13],1,Modbus_LabView_Data.InpRegisters_3xxx[15])SWPB(ModbusTCPIP_Data_SWPB[13],REVERSE,ModbusTCPIP:O.Data[15]);
   16: MUL(IO_Point_EX:7:I.Ch03.Data,10,FVIR_TC[14])SUB(FVIR_TC[14],39,FVIR_TC[14])MUL(FVIR_TC[14],1,Modbus_LabView_Data.InpRegisters_3xxx[16])SWPB(ModbusTCPIP_Data_SWPB[14],REVERSE,ModbusTCPIP:O.Data[16]);
   17: MUL(IO_Point_EX:7:I.Ch04.Data,10,FVIR_TC[15])SUB(FVIR_TC[15],20,FVIR_TC[15])MUL(FVIR_TC[15],1,Modbus_LabView_Data.InpRegisters_3xxx[17])SWPB(ModbusTCPIP_Data_SWPB[15],REVERSE,ModbusTCPIP:O.Data[17]);
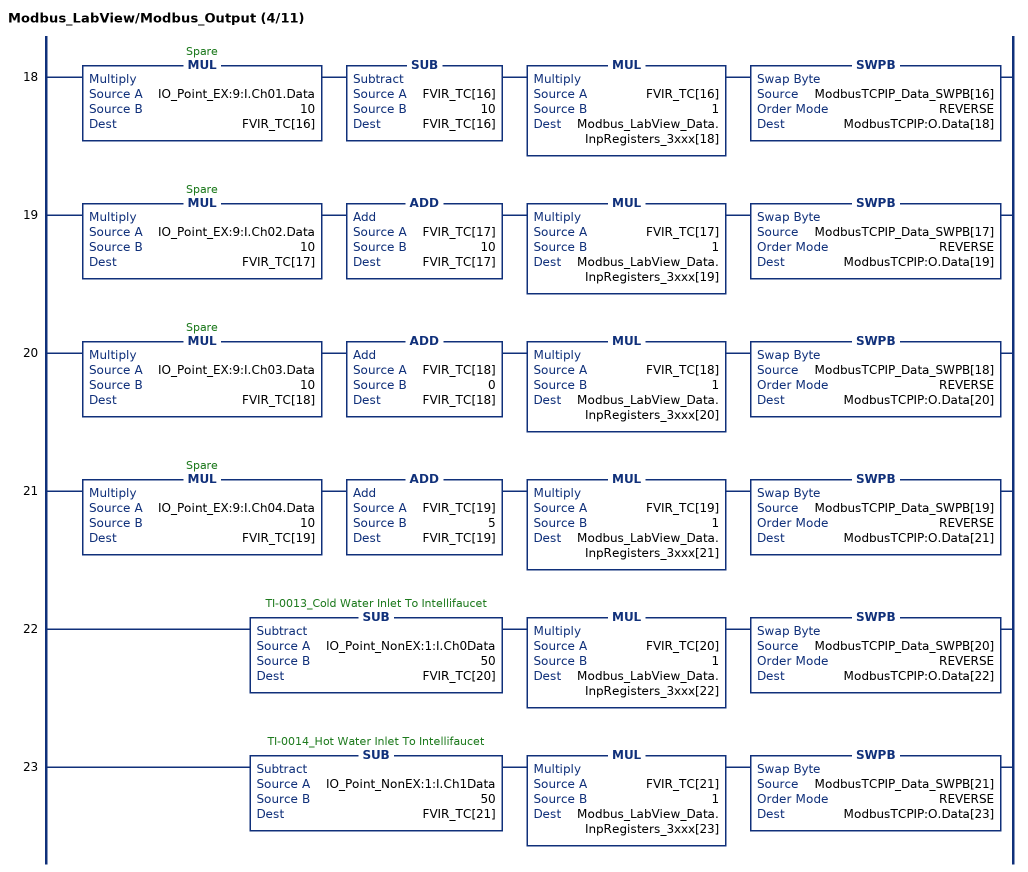
   18: MUL(IO_Point_EX:9:I.Ch01.Data,10,FVIR_TC[16])SUB(FVIR_TC[16],10,FVIR_TC[16])MUL(FVIR_TC[16],1,Modbus_LabView_Data.InpRegisters_3xxx[18])SWPB(ModbusTCPIP_Data_SWPB[16],REVERSE,ModbusTCPIP:O.Data[18]);
   19: MUL(IO_Point_EX:9:I.Ch02.Data,10,FVIR_TC[17])ADD(FVIR_TC[17],10,FVIR_TC[17])MUL(FVIR_TC[17],1,Modbus_LabView_Data.InpRegisters_3xxx[19])SWPB(ModbusTCPIP_Data_SWPB[17],REVERSE,ModbusTCPIP:O.Data[19]);
   20: MUL(IO_Point_EX:9:I.Ch03.Data,10,FVIR_TC[18])ADD(FVIR_TC[18],0,FVIR_TC[18])MUL(FVIR_TC[18],1,Modbus_LabView_Data.InpRegisters_3xxx[20])SWPB(ModbusTCPIP_Data_SWPB[18],REVERSE,ModbusTCPIP:O.Data[20]);
   21: MUL(IO_Point_EX:9:I.Ch04.Data,10,FVIR_TC[19])ADD(FVIR_TC[19],5,FVIR_TC[19])MUL(FVIR_TC[19],1,Modbus_LabView_Data.InpRegisters_3xxx[21])SWPB(ModbusTCPIP_Data_SWPB[19],REVERSE,ModbusTCPIP:O.Data[21]);
   22: SUB(IO_Point_NonEX:1:I.Ch0Data,50,FVIR_TC[20])MUL(FVIR_TC[20],1,Modbus_LabView_Data.InpRegisters_3xxx[22])SWPB(ModbusTCPIP_Data_SWPB[20],REVERSE,ModbusTCPIP:O.Data[22]);
   23: SUB(IO_Point_NonEX:1:I.Ch1Data,50,FVIR_TC[21])MUL(FVIR_TC[21],1,Modbus_LabView_Data.InpRegisters_3xxx[23])SWPB(ModbusTCPIP_Data_SWPB[21],REVERSE,ModbusTCPIP:O.Data[23]);
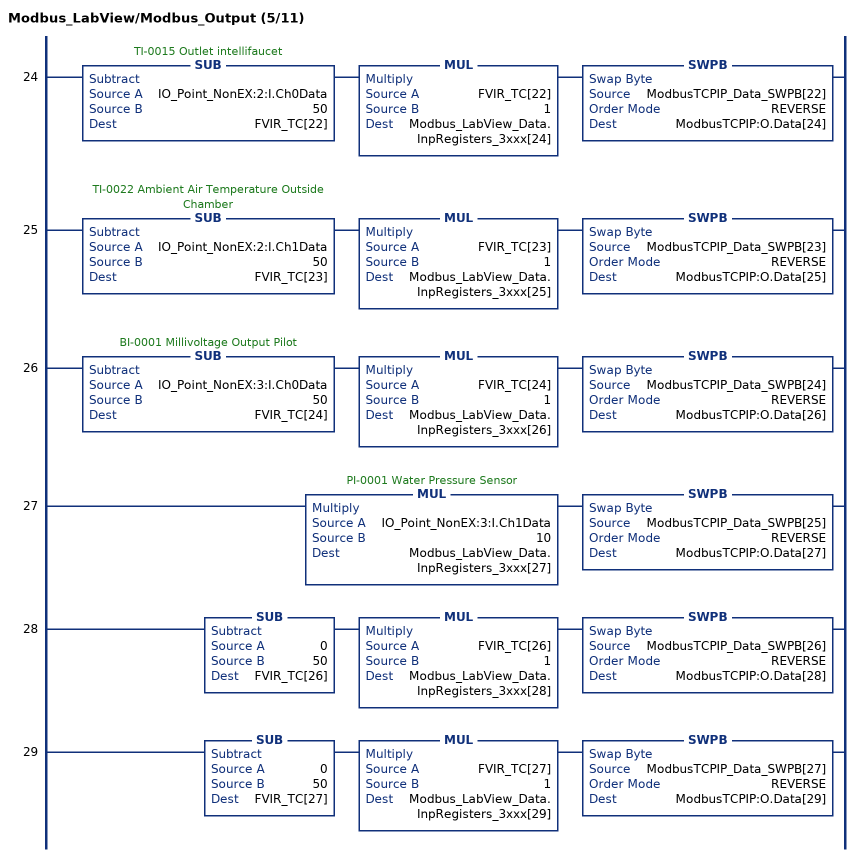
   24: SUB(IO_Point_NonEX:2:I.Ch0Data,50,FVIR_TC[22])MUL(FVIR_TC[22],1,Modbus_LabView_Data.InpRegisters_3xxx[24])SWPB(ModbusTCPIP_Data_SWPB[22],REVERSE,ModbusTCPIP:O.Data[24]);
   25: SUB(IO_Point_NonEX:2:I.Ch1Data,50,FVIR_TC[23])MUL(FVIR_TC[23],1,Modbus_LabView_Data.InpRegisters_3xxx[25])SWPB(ModbusTCPIP_Data_SWPB[23],REVERSE,ModbusTCPIP:O.Data[25]);
   26: SUB(IO_Point_NonEX:3:I.Ch0Data,50,FVIR_TC[24])MUL(FVIR_TC[24],1,Modbus_LabView_Data.InpRegisters_3xxx[26])SWPB(ModbusTCPIP_Data_SWPB[24],REVERSE,ModbusTCPIP:O.Data[26]);
   27: MUL(IO_Point_NonEX:3:I.Ch1Data,10,Modbus_LabView_Data.InpRegisters_3xxx[27])SWPB(ModbusTCPIP_Data_SWPB[25],REVERSE,ModbusTCPIP:O.Data[27]);
   28: SUB(0,50,FVIR_TC[26])MUL(FVIR_TC[26],1,Modbus_LabView_Data.InpRegisters_3xxx[28])SWPB(ModbusTCPIP_Data_SWPB[26],REVERSE,ModbusTCPIP:O.Data[28]);
   29: SUB(0,50,FVIR_TC[27])MUL(FVIR_TC[27],1,Modbus_LabView_Data.InpRegisters_3xxx[29])SWPB(ModbusTCPIP_Data_SWPB[27],REVERSE,ModbusTCPIP:O.Data[29]);
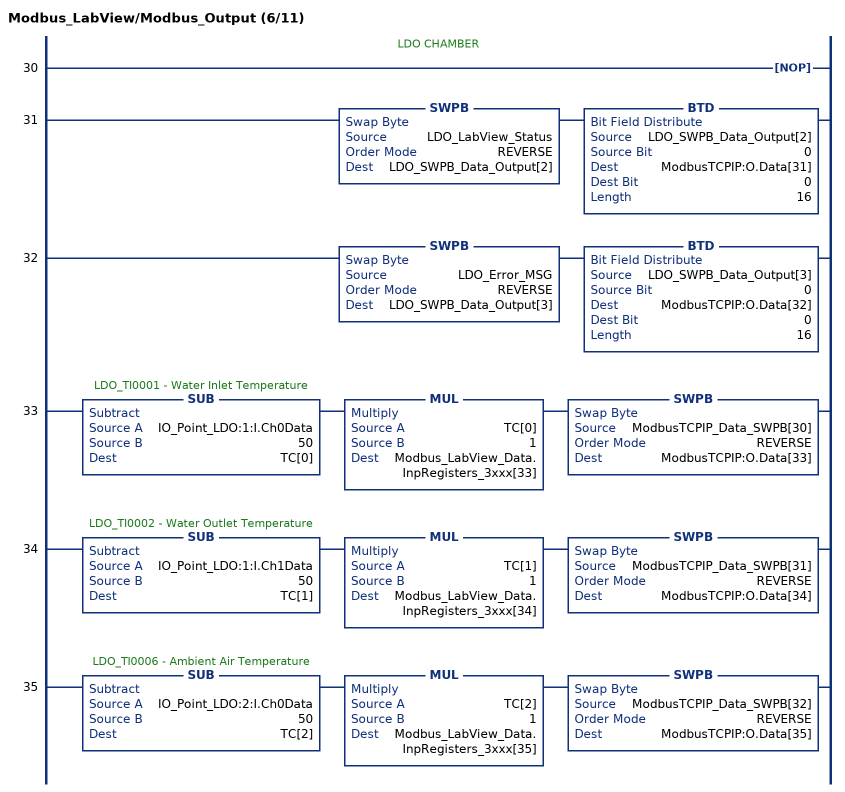
   // LDO CHAMBER
   30: NOP();
   31: SWPB(LDO_LabView_Status,REVERSE,LDO_SWPB_Data_Output[2])BTD(LDO_SWPB_Data_Output[2],0,ModbusTCPIP:O.Data[31],0,16);
   32: SWPB(LDO_Error_MSG,REVERSE,LDO_SWPB_Data_Output[3])BTD(LDO_SWPB_Data_Output[3],0,ModbusTCPIP:O.Data[32],0,16);
   33: SUB(IO_Point_LDO:1:I.Ch0Data,50,TC[0])MUL(TC[0],1,Modbus_LabView_Data.InpRegisters_3xxx[33])SWPB(ModbusTCPIP_Data_SWPB[30],REVERSE,ModbusTCPIP:O.Data[33]);
   34: SUB(IO_Point_LDO:1:I.Ch1Data,50,TC[1])MUL(TC[1],1,Modbus_LabView_Data.InpRegisters_3xxx[34])SWPB(ModbusTCPIP_Data_SWPB[31],REVERSE,ModbusTCPIP:O.Data[34]);
   35: SUB(IO_Point_LDO:2:I.Ch0Data,50,TC[2])MUL(TC[2],1,Modbus_LabView_Data.InpRegisters_3xxx[35])SWPB(ModbusTCPIP_Data_SWPB[32],REVERSE,ModbusTCPIP:O.Data[35]);
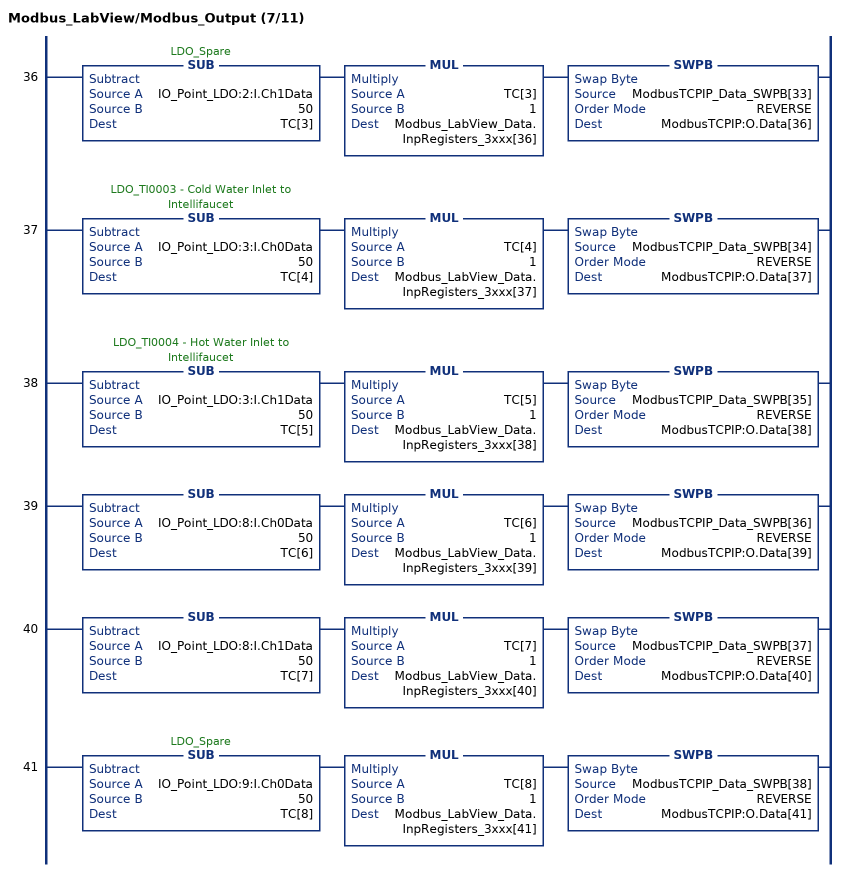
   36: SUB(IO_Point_LDO:2:I.Ch1Data,50,TC[3])MUL(TC[3],1,Modbus_LabView_Data.InpRegisters_3xxx[36])SWPB(ModbusTCPIP_Data_SWPB[33],REVERSE,ModbusTCPIP:O.Data[36]);
   37: SUB(IO_Point_LDO:3:I.Ch0Data,50,TC[4])MUL(TC[4],1,Modbus_LabView_Data.InpRegisters_3xxx[37])SWPB(ModbusTCPIP_Data_SWPB[34],REVERSE,ModbusTCPIP:O.Data[37]);
   38: SUB(IO_Point_LDO:3:I.Ch1Data,50,TC[5])MUL(TC[5],1,Modbus_LabView_Data.InpRegisters_3xxx[38])SWPB(ModbusTCPIP_Data_SWPB[35],REVERSE,ModbusTCPIP:O.Data[38]);
   39: SUB(IO_Point_LDO:8:I.Ch0Data,50,TC[6])MUL(TC[6],1,Modbus_LabView_Data.InpRegisters_3xxx[39])SWPB(ModbusTCPIP_Data_SWPB[36],REVERSE,ModbusTCPIP:O.Data[39]);
   40: SUB(IO_Point_LDO:8:I.Ch1Data,50,TC[7])MUL(TC[7],1,Modbus_LabView_Data.InpRegisters_3xxx[40])SWPB(ModbusTCPIP_Data_SWPB[37],REVERSE,ModbusTCPIP:O.Data[40]);
   41: SUB(IO_Point_LDO:9:I.Ch0Data,50,TC[8])MUL(TC[8],1,Modbus_LabView_Data.InpRegisters_3xxx[41])SWPB(ModbusTCPIP_Data_SWPB[38],REVERSE,ModbusTCPIP:O.Data[41]);
